// TIA Portal V20 export
TYPE "LER_PMC_Input_Data"
// stored: Access Published
   STRUCT
      Machining_Assembly : Struct   // Machining and Assembly
         FTQ_AllData_Rdy : Bool;   // FTQ All Data Ready
         FTQ_Data_Reset : Bool;   // FTQ Data Reset
         Buffer_Bypass : Bool;   // Buffer Bypass
         Bypassed : Bool;   // Bypassed
         CheckSum_OK : Bool;   // CheckSum OK
         PUNData_command : Bool;
         PUNData : String[20];   // PUN Data
         FTQ_PUNData : String[20];   // FTQ PUN Data
         GM_PartNumber : String[8];   // GM Part Number
         OptionalData : String[12];   // Optional Data
         PartTypeString : String[12];   // Part Type String
         FTQ_Reject_String : String[100];   // FTQ Reject String
         IncrGood_Count : Bool;   // Increment Good Count
         IncrReject_Count : Bool;   // Increment Reject Count
         Machine_Loading : Bool;   // Machine Loading
         Machine_Unloading : Bool;   // Machine Unloading
         Bypass_PartPallet_Inc : Bool;   // Bypass Part Pallet Increment
         Part_Type : Int;   // Part Type Integer
         Buffer_Count : Int;   // Buffer Count
         FTQ_Reject_Code : DInt;   // FTQ Reject Code
         Material_Low : Bool;   // Material Low / (See definition)
         AutoCycle_Running : Bool;   // AutoCycle Running
         ManualMode : Bool;   // Manual Mode
         Cycle_Time_Ready : Bool;   // Cycle Time Ready
         OperatorOvercycle_1 : Bool;   // Operator Overcycle 1
         OperatorOvercycle_2 : Bool;   // Operator Overcycle 2
         Blocked : Bool;   // Blocked
         Starved : Bool;   // Starved
         Idle : Bool;   // Idle
         Wait_1 : Bool;   // Wait 1
         Wait_2 : Bool;   // Wait 2
         Wait_3 : Bool;   // Wait 3
         Wait_4 : Bool;   // Wait 4
         Stopped_by_Operator : Bool;   // Stopped by Operator
         Machine_FaultedLevel1 : Bool;   // Machine Fault
         Machine_FaultedLevel2 : Bool;   // Machine Fault
         Machine_Fault : Bool;   // Machine Fault
         Fault_Ack : Bool;   // Fault Ack
         Quality_Check_Warning : Bool;   // Quality Check Warning
         Quality_Check_Fault : Bool;   // Quality Check Fault
         Quality_Ack : Bool;   // Quality Ack
         ToolChange_Warning : Bool;   // Tool Change Warning
         ToolChange_Fault : Bool;   // Tool Change Fault
         ToolChange_Ack_Action : Bool;   // Tool Change Ack
         Andon_Hold : Bool;   // Andon Hold
         Fault_Word : DInt;   // Fault Word
         Fault_String : String[200];   // Fault String
         Dry_Cycle_Mode : Bool;   // Dry Cycle Mode
         ControlPowerON : Bool;   // Control Power ON
         All_Maps_Out_Of_Auto : Bool;   // All Maps Out Of Auto
         No_Maps_Show_Fault : Bool;   // No Maps Show Fault
      END_STRUCT;
      Filter_Coolant : Struct   // Filter and Coolant
         Current_Temperature : Int;   // Current Temperature
         Numerical_Quan_1 : Int;   // Numerical Quantity 1
         Numerical_Quan_2 : Int;   // Numerical Quantity 2
         Numerical_Quan_3 : Int;   // Numerical Quantity 3
         Machine_Minor_Fault : Bool;   // Machine Minor Fault
         Tank_Coolant_Temp_OK : Bool;   // Tank Coolant Temp OK
         Tank_Coolant_Temp_HI : Bool;   // Tank Coolant Temp HI
         Tank_Coolant_Temp_Low : Bool;   // Tank Coolant Temp Low
         Tank_Lvl_OK : Bool;   // Tank Level OK
         Tank_Lvl_High : Bool;   // Tank Level High
         Tank_Lvl_Low : Bool;   // Tank Level Low
         Pump_Back_Lvl_OK : Bool;   // Pump Back Level OK
         Pump_Back_Lvl_High : Bool;   // Pump Back Level High
         Pump_Back_Lvl_Low : Bool;   // Pump Back Level Low
      END_STRUCT;
      CMM : Struct   // CMM
         Bad_Quality_Data : Bool;   // Bad Quality Data
         No_Queue_Avail : Bool;   // No Queue Available
         Queue_Avail : Bool;   // Queue Available
         Insp_Prog_Running : Bool;   // Inspection Program Running
         Time_Remailing : Int;   // Time Remailing
      END_STRUCT;
   END_STRUCT;
END_TYPE
